(* Logix 5000 project; controller Primary vendor 1 type 14 code 196 rev 37.11; software revision 37.00; part 2 of 2 *)
(* tags used below, declared in another part *)
   DINT : DINT;
   HMI_Cmd : Hot_Backup_HMI_Interface;
   HMI_Event_Log : Hot_Backup_Event_Log[10];
   HMI_Handshake : Hot_Backup_HMI_Interface;
   Manual_Switchover_PB : BOOL;
   PEER_HB_Consume : Hot_Backup_Interface;   // Consumed data from the parter controller
   PEER_HB_Produce : Hot_Backup_Interface;   // Produced data to the peer controller.

PROGRAM Hot_Backup   (* main routine AOI_CALL *)
VAR
   Hot_Backup : Hot_Backup := (Sts_OutputsFaulted := 1, Sts_PeerReady := 1, Sts_Primary := 1);   // SoS AOI Tag Structure
   ONS : DINT;   // Bits are reserved for One Shots
   Sts_FirstScanBit : BOOL := 1;   // Set to "1" when the first scan bit is set.
   Sts_OutputsFaulted : BOOL := 1;   // Set to "1" when all output modules are faulted
   Sts_OutputsInhibited : BOOL;   // Set to "1" when all output modules are Inhibited
   Sts_OutputsRunning : BOOL;   // Set to "1" when all output modules are running
   Val_ModuleEntryStatus : DINT := 12288;   // This word contains the module entry status for each gsv.
   Val_ModuleMode : DINT;   // This word contains the module mode status for each gsv/ssv.
   Val_OutputsFaulted : DINT[2];   // These words will be a non zero value if any output module is faulted.
   Val_OutputsInhibited : DINT[2];   // These words will be a non zero value if any output module is inhibited.
   Val_OutputsRunning : DINT[2];   // These words will be a non zero value if any output module is running.
   Val_OutputsWaiting : DINT[2] := ([0] := 1);   // These words will be a non zero value if any output module is waiting.
END_VAR

ROUTINE AOI_CALL   (* ladder *)
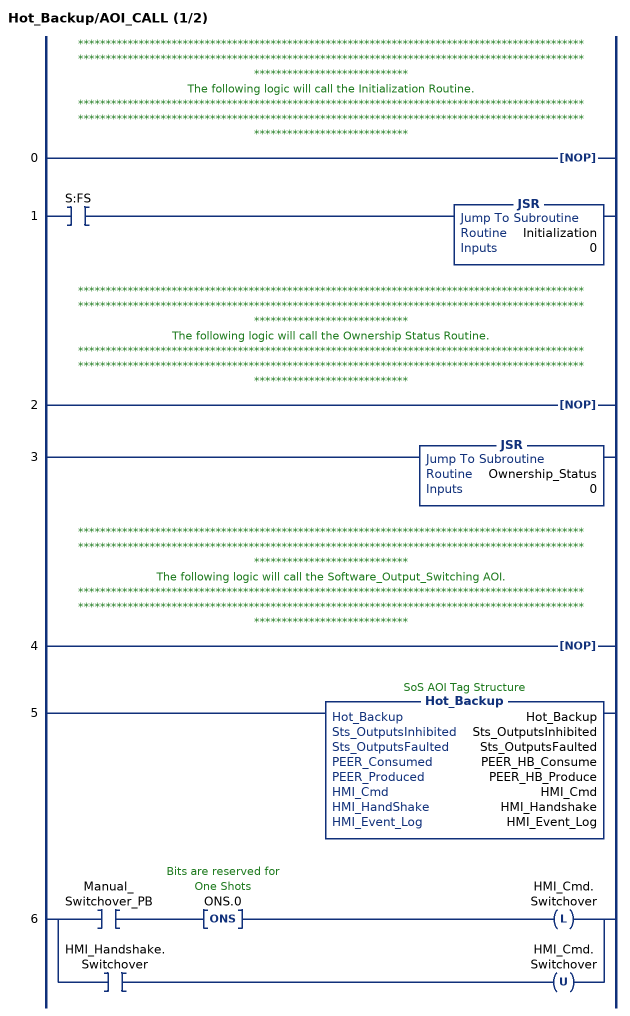
   // ********************************************************************************************************************************************************************************************************************
   // The following logic will call the Initialization Routine.
   // ********************************************************************************************************************************************************************************************************************
   0: NOP();
   1: XIC(S:FS)JSR(Initialization,0);
   // ********************************************************************************************************************************************************************************************************************
   // The following logic will call the Ownership Status Routine.
   // ********************************************************************************************************************************************************************************************************************
   2: NOP();
   3: JSR(Ownership_Status,0);
   // ********************************************************************************************************************************************************************************************************************
   // The following logic will call the Software_Output_Switching AOI.
   // ********************************************************************************************************************************************************************************************************************
   4: NOP();
   5: Hot_Backup(Hot_Backup,Sts_OutputsInhibited,Sts_OutputsFaulted,PEER_HB_Consume,PEER_HB_Produce,HMI_Cmd,HMI_Handshake,HMI_Event_Log);
   6: [XIC(Manual_Switchover_PB) ONS(ONS.0) OTL(HMI_Cmd.Switchover) ,XIC(HMI_Handshake.Switchover) OTU(HMI_Cmd.Switchover) ];
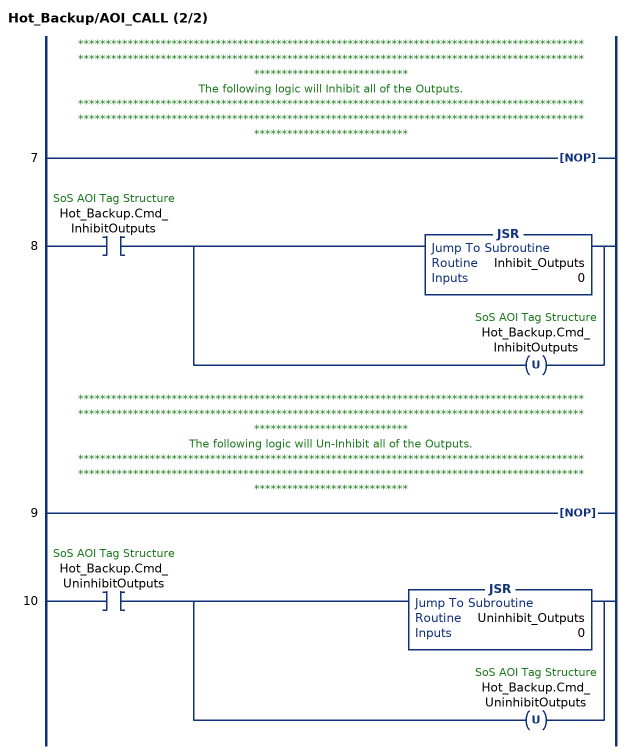
   // ********************************************************************************************************************************************************************************************************************
   // The following logic will Inhibit all of the Outputs.
   // ********************************************************************************************************************************************************************************************************************
   7: NOP();
   8: XIC(Hot_Backup.Cmd_InhibitOutputs)[JSR(Inhibit_Outputs,0) ,OTU(Hot_Backup.Cmd_InhibitOutputs) ];
   // ********************************************************************************************************************************************************************************************************************
   // The following logic will Un-Inhibit all of the Outputs.
   // ********************************************************************************************************************************************************************************************************************
   9: NOP();
   10: XIC(Hot_Backup.Cmd_UninhibitOutputs)[JSR(Uninhibit_Outputs,0) ,OTU(Hot_Backup.Cmd_UninhibitOutputs) ];
END_ROUTINE

ROUTINE Inhibit_Outputs   (* ladder *)
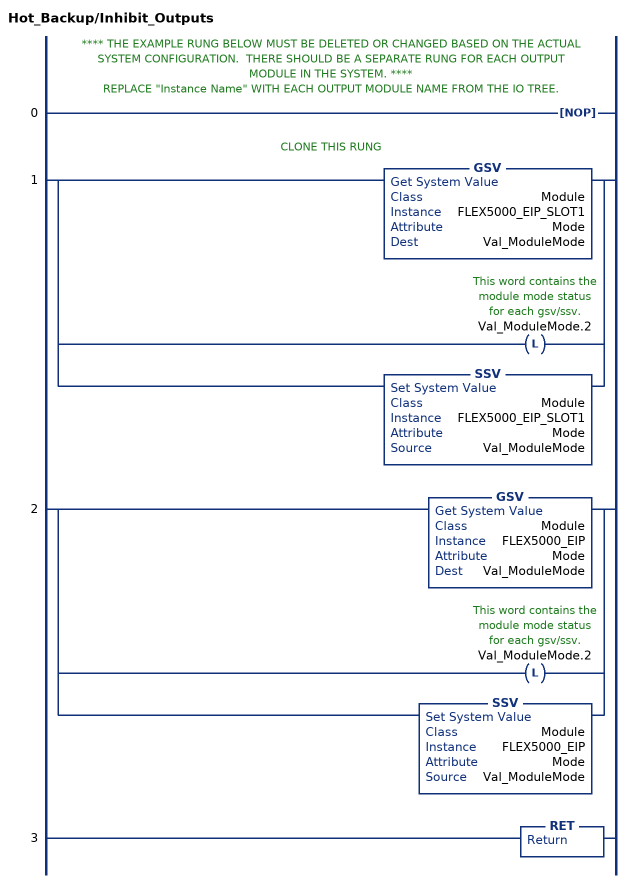
   // **** THE EXAMPLE RUNG BELOW MUST BE DELETED OR CHANGED BASED ON THE ACTUAL SYSTEM CONFIGURATION.  THERE SHOULD BE A SEPARATE RUNG FOR EACH OUTPUT MODULE IN THE SYSTEM. ****
   // REPLACE "Instance Name" WITH EACH OUTPUT MODULE NAME FROM THE IO TREE.
   0: NOP();
   // CLONE THIS RUNG
   1: [GSV(Module,FLEX5000_EIP_SLOT1,Mode,Val_ModuleMode) ,OTL(Val_ModuleMode.2) ,SSV(Module,FLEX5000_EIP_SLOT1,Mode,Val_ModuleMode) ];
   2: [GSV(Module,FLEX5000_EIP,Mode,Val_ModuleMode) ,OTL(Val_ModuleMode.2) ,SSV(Module,FLEX5000_EIP,Mode,Val_ModuleMode) ];
   3: RET();
END_ROUTINE

ROUTINE Initialization   (* ladder *)
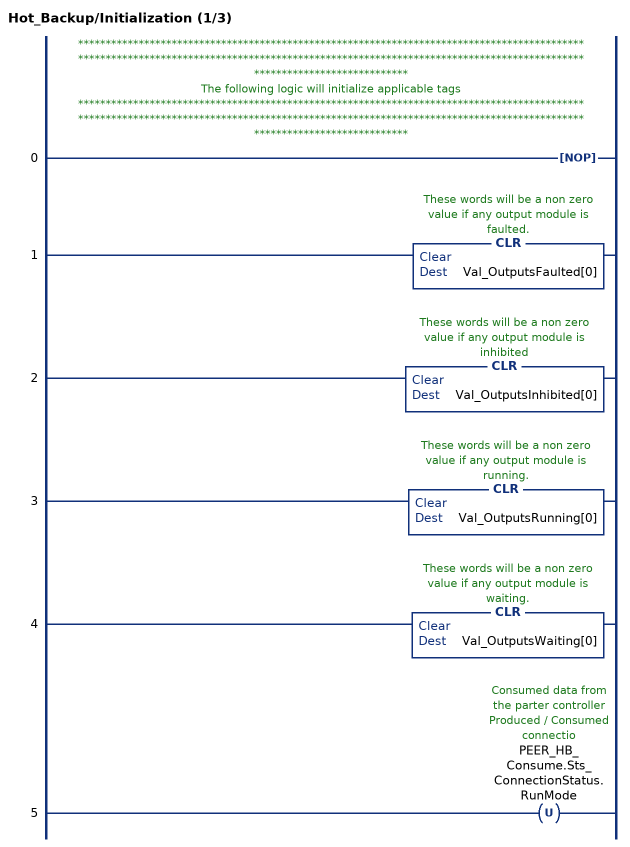
   // ********************************************************************************************************************************************************************************************************************
   // The following logic will initialize applicable tags
   // ********************************************************************************************************************************************************************************************************************
   0: NOP();
   1: CLR(Val_OutputsFaulted[0]);
   2: CLR(Val_OutputsInhibited[0]);
   3: CLR(Val_OutputsRunning[0]);
   4: CLR(Val_OutputsWaiting[0]);
   5: OTU(PEER_HB_Consume.Sts_ConnectionStatus.RunMode);
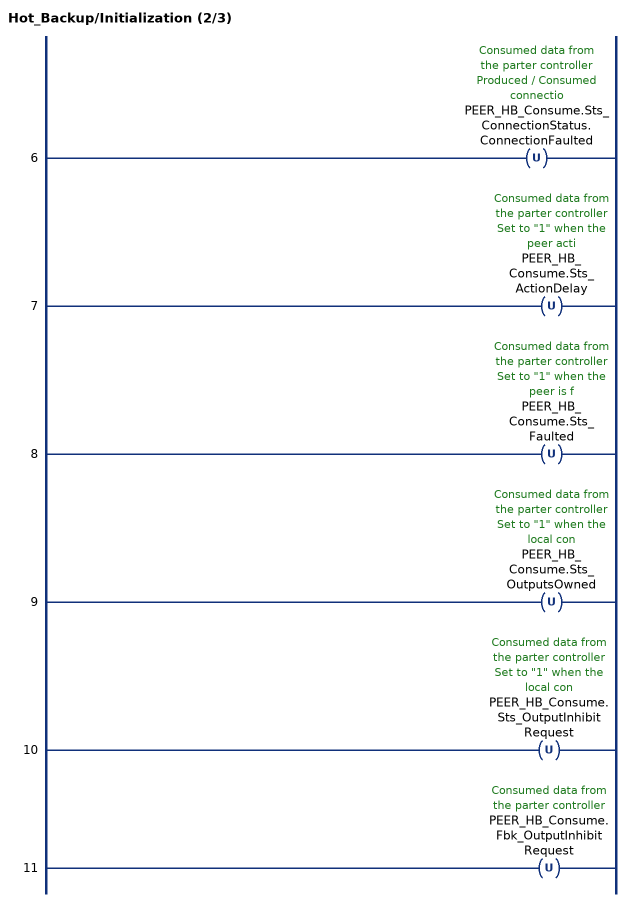
   6: OTU(PEER_HB_Consume.Sts_ConnectionStatus.ConnectionFaulted);
   7: OTU(PEER_HB_Consume.Sts_ActionDelay);
   8: OTU(PEER_HB_Consume.Sts_Faulted);
   9: OTU(PEER_HB_Consume.Sts_OutputsOwned);
   10: OTU(PEER_HB_Consume.Sts_OutputInhibitRequest);
   11: OTU(PEER_HB_Consume.Fbk_OutputInhibitRequest);
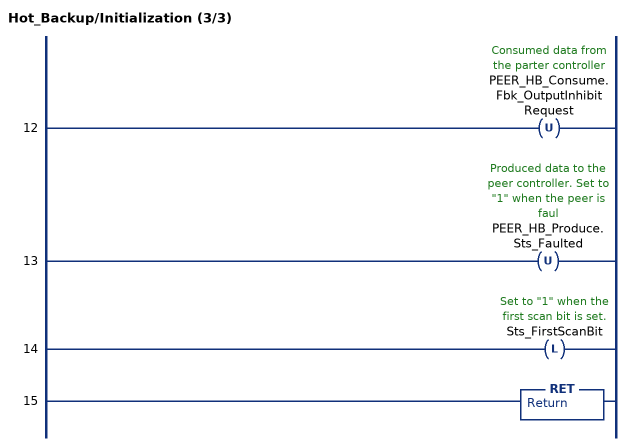
   12: OTU(PEER_HB_Consume.Fbk_OutputInhibitRequest);
   13: OTU(PEER_HB_Produce.Sts_Faulted);
   14: OTL(Sts_FirstScanBit);
   15: RET();
END_ROUTINE

ROUTINE Ownership_Status   (* ladder *)
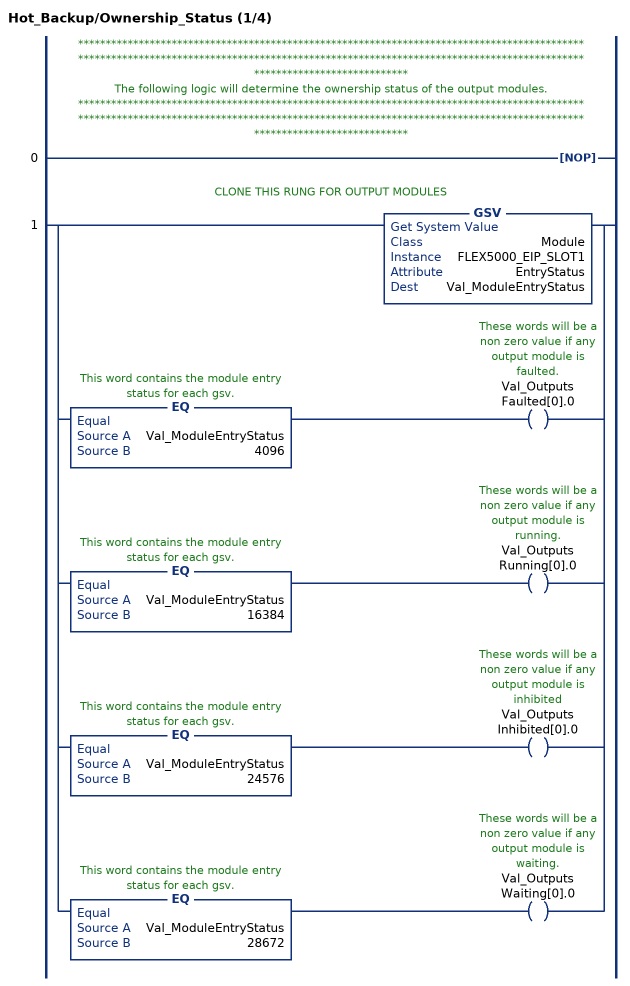
   // ********************************************************************************************************************************************************************************************************************
   // The following logic will determine the ownership status of the output modules.
   // ********************************************************************************************************************************************************************************************************************
   0: NOP();
   // CLONE THIS RUNG FOR OUTPUT MODULES
   1: [GSV(Module,FLEX5000_EIP_SLOT1,EntryStatus,Val_ModuleEntryStatus) ,EQ(Val_ModuleEntryStatus,4096) OTE(Val_OutputsFaulted[0].0) ,EQ(Val_ModuleEntryStatus,16384) OTE(Val_OutputsRunning[0].0) ,EQ(Val_ModuleEntryStatus,24576) OTE(Val_OutputsInhibited[0].0) ,EQ(Val_ModuleEntryStatus,28672) OTE(Val_OutputsWaiting[0].0) ];
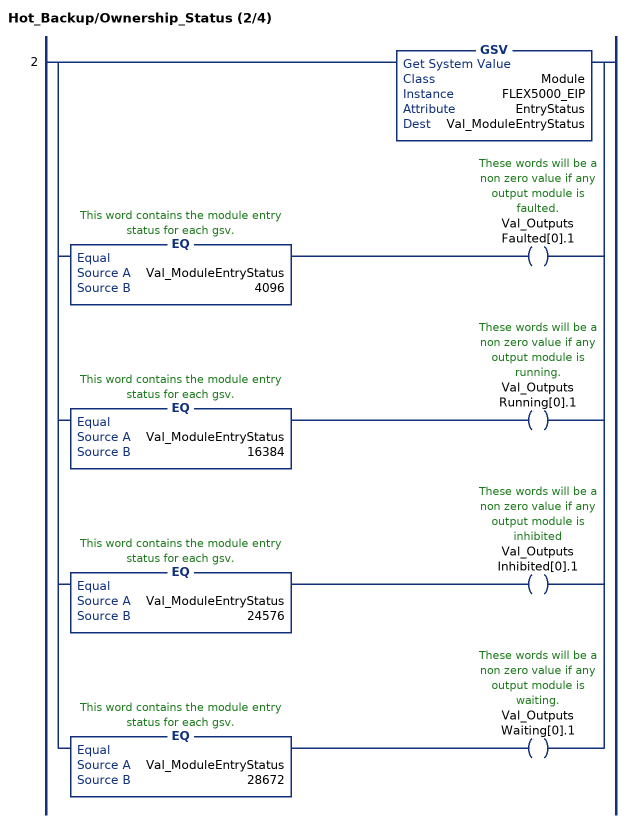
   2: [GSV(Module,FLEX5000_EIP,EntryStatus,Val_ModuleEntryStatus) ,EQ(Val_ModuleEntryStatus,4096) OTE(Val_OutputsFaulted[0].1) ,EQ(Val_ModuleEntryStatus,16384) OTE(Val_OutputsRunning[0].1) ,EQ(Val_ModuleEntryStatus,24576) OTE(Val_OutputsInhibited[0].1) ,EQ(Val_ModuleEntryStatus,28672) OTE(Val_OutputsWaiting[0].1) ];
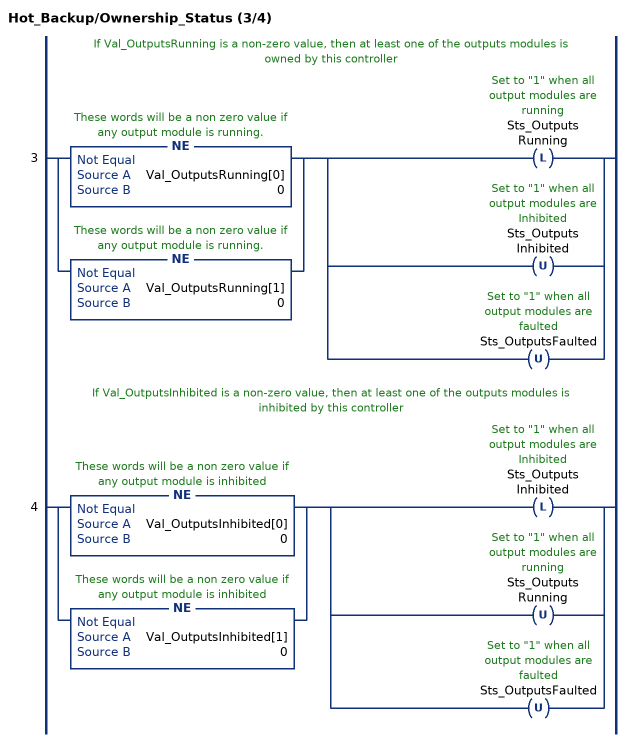
   // If Val_OutputsRunning is a non-zero value, then at least one of the outputs modules is owned by this controller
   3: [NE(Val_OutputsRunning[0],0) ,NE(Val_OutputsRunning[1],0) ][OTL(Sts_OutputsRunning) ,OTU(Sts_OutputsInhibited) ,OTU(Sts_OutputsFaulted) ];
   // If Val_OutputsInhibited is a non-zero value, then at least one of the outputs modules is inhibited by this controller
   4: [NE(Val_OutputsInhibited[0],0) ,NE(Val_OutputsInhibited[1],0) ][OTL(Sts_OutputsInhibited) ,OTU(Sts_OutputsRunning) ,OTU(Sts_OutputsFaulted) ];
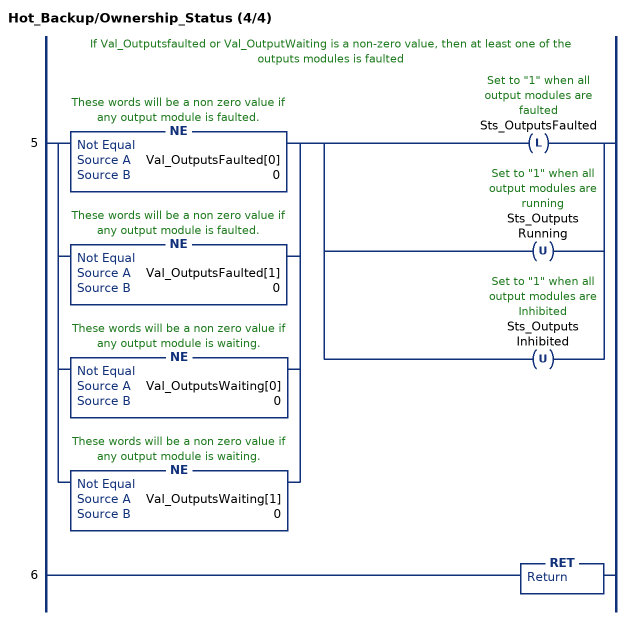
   // If Val_Outputsfaulted or Val_OutputWaiting is a non-zero value, then at least one of the outputs modules is faulted
   5: [NE(Val_OutputsFaulted[0],0) ,NE(Val_OutputsFaulted[1],0) ,NE(Val_OutputsWaiting[0],0) ,NE(Val_OutputsWaiting[1],0) ][OTL(Sts_OutputsFaulted) ,OTU(Sts_OutputsRunning) ,OTU(Sts_OutputsInhibited) ];
   6: RET();
END_ROUTINE

ROUTINE Uninhibit_Outputs   (* ladder *)
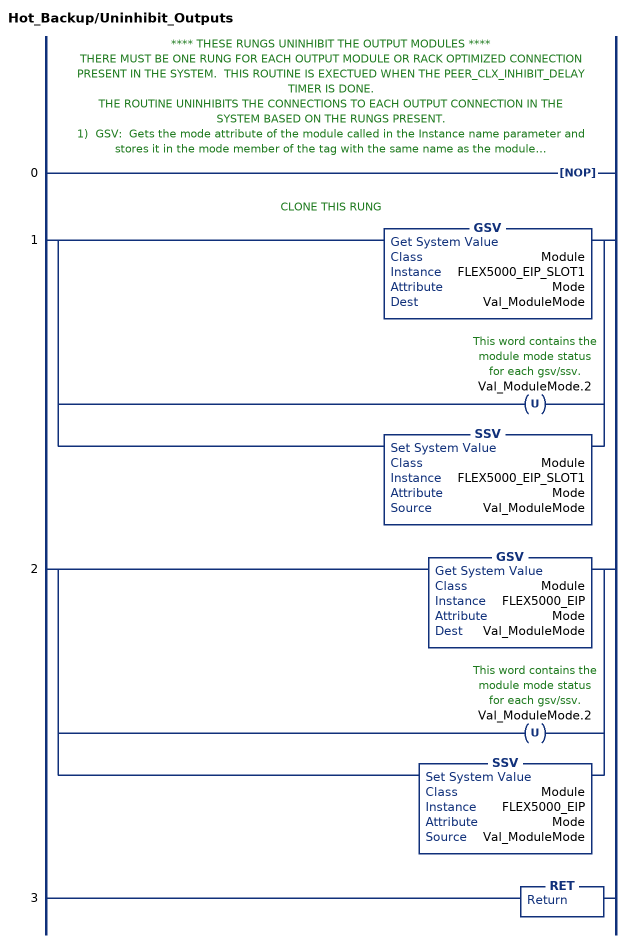
   // **** THESE RUNGS UNINHIBIT THE OUTPUT MODULES ****
   // THERE MUST BE ONE RUNG FOR EACH OUTPUT MODULE OR RACK OPTIMIZED CONNECTION PRESENT IN THE SYSTEM.  THIS ROUTINE IS EXECTUED WHEN THE PEER_CLX_INHIBIT_DELAY TIMER IS DONE.
   // THE ROUTINE UNINHIBITS THE CONNECTIONS TO EACH OUTPUT CONNECTION IN THE SYSTEM BASED ON THE RUNGS PRESENT.
   // 1)  GSV:  Gets the mode attribute of the module called in the Instance name parameter and stores it in the mode member of the tag with the same name as the module.
   // 2)  Clears bit 2 of the mode member, which indicates that the controller should uninhibit its connection to the module.
   // 3)  SSV: Sends the new mode value to the mode member of the tag with the same name as the module, which uninhibits that connection.
   // **** THE EXAMPLE RUNG BELOW MUST BE DELETED OR CHANGED BASED ON THE ACTUAL SYSTEM CONFIGURATION. ****
   // REPLACE "Source" WITH YOUR MODULE NAME FROM THE IO TREE.
   // - for each Comms Module in your system
   // - for each Output Module in your system
   0: NOP();
   // CLONE THIS RUNG
   1: [GSV(Module,FLEX5000_EIP_SLOT1,Mode,Val_ModuleMode) ,OTU(Val_ModuleMode.2) ,SSV(Module,FLEX5000_EIP_SLOT1,Mode,Val_ModuleMode) ];
   2: [GSV(Module,FLEX5000_EIP,Mode,Val_ModuleMode) ,OTU(Val_ModuleMode.2) ,SSV(Module,FLEX5000_EIP,Mode,Val_ModuleMode) ];
   3: RET();
END_ROUTINE
END_PROGRAM

PROGRAM MainProgram   (* main routine MainRoutine *)
VAR
   ProgramTag : DINT;
END_VAR

ROUTINE MainRoutine   (* ladder *)
END_ROUTINE
END_PROGRAM
